TYPE TTank :
STRUCT
	Mixer : TEngine;
	ValveFilling : TValve;
	ValveDraining : TValve;
	Heater : THeater;
	
	Filling : TPhaseFilling;
	Draining : TPhaseDraining;
	Mixing : TPhaseMixing;
	Heating : TPhaseHeating;
	
	GlobalError : BOOL;

END_STRUCT
END_TYPE

(* stored: Version 1.1.0.1, ProductVersion 3.1.4024.13
   DUT TTank: Id {8ca78818-1b53-487b-b198-f81c31206d49} *)
